TYPE ACRMemoryRealEvents :
STRUCT
	_Values : ARRAY [0..GCL.cMemoryEventsMAX] OF ACRMemoryRealEvent;
END_STRUCT
END_TYPE

(* stored: Version 1.1.0.1, ProductVersion 3.1.4020.12
   DUT ACRMemoryRealEvents: Id {7586dcdd-a760-4dee-8b72-c7ac49ff6596} *)
